(* IEC 61131-3 sources: AXOpen/src/abstractions/ctrl/src/Messaging/Dynamic, 9 files *)

(* ---- eAxoMessageDigestMethod.st ---- *)
NAMESPACE AXOpen.Messaging.Dynamic
    /// <summary>
    /// Message digest methods used to create fingerprint of a message.
    /// </summary>
    TYPE eAxoMessageDigestMethod : INT
    (
        /// <summary>
        /// Fastest method with highest probability of colisions.
        /// </summary>
        CRC8 := 8,

        /// <summary>
        /// Moderate speed method with lower probability of colisions.
        /// </summary>
        CRC16 := 16,

        /// <summary>
        /// Slowest speed method with relatively low probability of colisions.
        /// </summary>
        CRC32 := 32,

        /// <summary>
        /// Messages are not digested the repeated messages won't be filtered out.
        /// Use this option on low performance devices.
        /// </summary>
        NONE := 32767
    );
    END_TYPE
END_NAMESPACE

(* ---- IAxoMessageCategorize.st ---- *)
NAMESPACE AXOpen.Messaging.Dynamic
    INTERFACE IAxoMessageCategorize
		/// <summary>
        /// Categorizes and creates the message as 'debug'.
		/// </summary>
        METHOD AsDebug : IAxoMessageProperties END_METHOD

		/// <summary>
        /// Categorizes and creates the message as 'error'.
		/// </summary>
        METHOD AsError : IAxoMessageProperties END_METHOD

		/// <summary>
        /// Categorizes and creates the message as 'fatal'.
		/// </summary>
        METHOD AsFatal : IAxoMessageProperties END_METHOD

		/// <summary>
        /// Categorizes and creates the message as 'info'.
		/// </summary>
        METHOD AsInfo : IAxoMessageProperties END_METHOD

		/// <summary>
        /// Categorizes and creates the message as 'trace'.
		/// </summary>
        METHOD AsTrace : IAxoMessageProperties END_METHOD

		/// <summary>
        /// Categorizes and creates the message as 'warning'.
		/// </summary>
        METHOD AsWarning : IAxoMessageProperties END_METHOD
    END_INTERFACE
END_NAMESPACE

(* ---- IAxoMessageProperties.st ---- *)
NAMESPACE AXOpen.Messaging.Dynamic
    INTERFACE IAxoMessageProperties
        METHOD Pin: IAxoMessageProperties END_METHOD
        METHOD IsPinned: BOOL END_METHOD
    END_INTERFACE
END_NAMESPACE

(* ---- IAxoMessages.st ---- *)
NAMESPACE AXOpen.Messaging.Dynamic
    INTERFACE IAxoMessages
	    /// <summary>
		/// Adds message of 'debug' category to the message queue.
		/// </summary>
        METHOD Debug : IAxoMessageProperties
            VAR_INPUT
                /// <summary>
                /// Arbitrary message string.
                /// </summary>
                Message : STRING[AxoIntConstants#MAX_MESSAGE_TEXT_LENGHT];
            END_VAR
        END_METHOD

	    /// <summary>
		/// Adds message of 'error' category to the message queue.
		/// </summary>
        METHOD Error : IAxoMessageProperties
            VAR_INPUT
                /// <summary>
                /// Arbitrary message string.
                /// </summary>
                Message : STRING[AxoIntConstants#MAX_MESSAGE_TEXT_LENGHT];
            END_VAR
        END_METHOD

	    /// <summary>
		/// Adds message of 'information' category to the message queue.
		/// </summary>
        METHOD Info : IAxoMessageProperties
            VAR_INPUT
                /// <summary>
                /// Arbitrary message string.
                /// </summary>
                Message : STRING[AxoIntConstants#MAX_MESSAGE_TEXT_LENGHT];
            END_VAR
        END_METHOD

	    /// <summary>
		/// Adds message of 'notification' category to the message queue.
		/// </summary>
        METHOD Notify : IAxoMessageProperties
            VAR_INPUT
                /// <summary>
                /// Arbitrary message string.
                /// </summary>
                Message : STRING[AxoIntConstants#MAX_MESSAGE_TEXT_LENGHT];
            END_VAR
        END_METHOD

	    /// <summary>
		/// Adds message of 'programming error' category to the message queue.
		/// </summary>
        METHOD Programming : IAxoMessageProperties
            VAR_INPUT
                /// <summary>
                /// Arbitrary message string.
                /// </summary>
                Message : STRING[AxoIntConstants#MAX_MESSAGE_TEXT_LENGHT];
            END_VAR
        END_METHOD

	    /// <summary>
		/// Adds message of 'trace' category to the message queue.
		/// </summary>
        METHOD Trace : IAxoMessageProperties
            VAR_INPUT
                /// <summary>
                /// Arbitrary message string.
                /// </summary>
                Message : STRING[AxoIntConstants#MAX_MESSAGE_TEXT_LENGHT];
            END_VAR
        END_METHOD

	    /// <summary>
		/// Adds message of 'warning' category to the message queue.
		/// </summary>
        METHOD Warning : IAxoMessageProperties
            VAR_INPUT
                /// <summary>
                /// Arbitrary message string.
                /// </summary>
                Message : STRING[AxoIntConstants#MAX_MESSAGE_TEXT_LENGHT];
            END_VAR
        END_METHOD

        METHOD Build: IAxoMessageTextBuilder END_METHOD

        /// <summary>
		/// Adds message of given category to the message queue.
		/// </summary>
		/// <returns>Message index.</returns>
        METHOD Post  : IAxoMessageProperties
            VAR_INPUT
                /// <summary>
                /// Arbitrary message string.
                /// </summary>
                Message : STRING[AxoIntConstants#MAX_MESSAGE_TEXT_LENGHT];
                /// <summary>
                /// Message category.
                /// </summary>
                Category : eAxoMessageCategory;
            END_VAR
        END_METHOD

		/// <summary>
		/// Unpins this messenger.
		/// </summary>
        METHOD UnPin END_METHOD

    END_INTERFACE
END_NAMESPACE

(* ---- IAxoMessageTextBuilder.st ---- *)
NAMESPACE AXOpen.Messaging.Dynamic
    INTERFACE IAxoMessageTextBuilder
		/// <summary>
		/// Appends string to the message text.
		/// </summary>
		/// <remarks>
		/// 	<note type="warning">
		/// 		The size of the resulting string should not be more than '160' characters. The characters exceeding this size will be truncated.
		/// 	</note>
		/// </remarks>
 		METHOD Append : IAxoMessageTextBuilder VAR_INPUT Data : BOOL; END_VAR END_METHOD
		METHOD Append : IAxoMessageTextBuilder VAR_INPUT Data : BYTE; END_VAR END_METHOD
		METHOD Append : IAxoMessageTextBuilder VAR_INPUT Data : WORD; END_VAR END_METHOD
		METHOD Append : IAxoMessageTextBuilder VAR_INPUT Data : DWORD; END_VAR END_METHOD
		METHOD Append : IAxoMessageTextBuilder VAR_INPUT Data : LWORD; END_VAR END_METHOD
		METHOD Append : IAxoMessageTextBuilder VAR_INPUT Data : SINT; END_VAR END_METHOD
		METHOD Append : IAxoMessageTextBuilder VAR_INPUT Data : INT; END_VAR END_METHOD
		METHOD Append : IAxoMessageTextBuilder VAR_INPUT Data : DINT; END_VAR END_METHOD
		METHOD Append : IAxoMessageTextBuilder VAR_INPUT Data : LINT; END_VAR END_METHOD
		METHOD Append : IAxoMessageTextBuilder VAR_INPUT Data : USINT; END_VAR END_METHOD
		METHOD Append : IAxoMessageTextBuilder VAR_INPUT Data : UINT; END_VAR END_METHOD
		METHOD Append : IAxoMessageTextBuilder VAR_INPUT Data : UDINT; END_VAR END_METHOD
		METHOD Append : IAxoMessageTextBuilder VAR_INPUT Data : ULINT; END_VAR END_METHOD
		METHOD Append : IAxoMessageTextBuilder VAR_INPUT Data : REAL; END_VAR END_METHOD
		METHOD Append : IAxoMessageTextBuilder VAR_INPUT Data : LREAL; END_VAR END_METHOD
		METHOD Append : IAxoMessageTextBuilder VAR_INPUT Data : TIME; END_VAR END_METHOD
		METHOD Append : IAxoMessageTextBuilder VAR_INPUT Data : LTIME; END_VAR END_METHOD
		METHOD Append : IAxoMessageTextBuilder VAR_INPUT Data : DATE; END_VAR END_METHOD
		METHOD Append : IAxoMessageTextBuilder VAR_INPUT Data : LDATE; END_VAR END_METHOD
		METHOD Append : IAxoMessageTextBuilder VAR_INPUT Data : TIME_OF_DAY; END_VAR END_METHOD
		METHOD Append : IAxoMessageTextBuilder VAR_INPUT Data : LTIME_OF_DAY; END_VAR END_METHOD
		METHOD Append : IAxoMessageTextBuilder VAR_INPUT Data : DATE_AND_TIME; END_VAR END_METHOD
		METHOD Append : IAxoMessageTextBuilder VAR_INPUT Data : LDATE_AND_TIME; END_VAR END_METHOD
		METHOD Append : IAxoMessageTextBuilder VAR_INPUT Data : CHAR; END_VAR END_METHOD
		// METHOD Append : IAxoMessageTextBuilder VAR_INPUT Data : WCHAR; END_VAR END_METHOD
		METHOD Append : IAxoMessageTextBuilder VAR_INPUT Data : STRING[AxoIntConstants#MAX_MESSAGE_TEXT_LENGHT]; END_VAR END_METHOD
		// METHOD Append : IAxoMessageTextBuilder VAR_INPUT Data : WSTRING[IxIntConstants#MAX_MESSAGE_TEXT_LENGHT]; END_VAR END_METHOD
		/// <summary>
		/// Gets categorization methods for fluent message builder.
		/// </summary>
        METHOD As : IAxoMessageCategorize END_METHOD

		/// <summary>
		/// Initiates new message text building for this messenger in fluent-like fashion.
		/// </summary>
        METHOD Build : IAxoMessageTextBuilder END_METHOD
    END_INTERFACE
END_NAMESPACE

(* ---- IAxoMessenger.st ---- *)
NAMESPACE AXOpen.Messaging.Dynamic
    INTERFACE IAxoMessenger
		/// <summary>
		/// Clears the message content.
		/// <remarks>
		/// 	<note type="important">
		/// 		This method is exposed for Rpc calls, for testing purposes. Rpc calls of this method must not be used in production code
		///		</note>
		/// </remarks>
		/// </summary>
		METHOD Clear END_METHOD

		METHOD OnCondition : IAxoMessages
			VAR_INPUT
				inCondition : BOOL;
			END_VAR
		END_METHOD
    END_INTERFACE
END_NAMESPACE

(* ---- IAxoMessengerEnv.st ---- *)
NAMESPACE AXOpen.Messaging.Dynamic
    INTERFACE IAxoMessengerEnv
		/// <summary>
		/// Gets whether the messaging is suspended at this point in program.
		/// <para>
		/// See also <see cref="PlcDocu.TcoCore.TcoMessengerSettings.Resume()"/>
		/// </para>
		/// <para>
		/// See also <see cref="PlcDocu.TcoCore.TcoMessengerSettings.Suspend()"/>
		/// </para>
		/// <para>
		/// See also <see cref="PlcDocu.TcoCore.TcoMessengerSettings.MinLevel"/>
		/// </para>
		/// </summary>
		METHOD IsSuspended: BOOL END_METHOD
		/// <summary>
		/// Gets the message digest method.
		/// Message digest serves to fingerprint messages.
		/// </summary>
		METHOD GetMessageDigestMethod : eAxoMessageDigestMethod END_METHOD
		/// <summary>
		/// Sets the message digest method.
		/// Message digest serves to fingerprint messages.
		/// </summary>
		METHOD SetMessageDigestMethod VAR_INPUT inDigestMethod : eAxoMessageDigestMethod; END_VAR END_METHOD
		/// <summary>
		/// Gets the minimal messaging level, the objects will post only messages for the levels of this or superior severity.
		/// <para>
		/// See also <see cref="PlcDocu.TcoCore.TcoMessengerSettings.Resume()"/>
		/// </para>
		/// <para>
		/// See also <see cref="PlcDocu.TcoCore.TcoMessengerSettings.Suspend()"/>
		/// </para>
		/// <para>
		/// See also <see cref="PlcDocu.TcoCore.TcoMessengerSettings.MinLevel"/>
		/// </para>
		/// </summary>
		METHOD GetMinLevel : eAxoMessageCategory END_METHOD
		/// <summary>
		/// Sets the minimal messaging level, the objects will post only messages for the levels of this or superior severity.
		/// <para>
		/// See also <see cref="PlcDocu.TcoCore.TcoMessengerSettings.Resume()"/>
		/// </para>
		/// <para>
		/// See also <see cref="PlcDocu.TcoCore.TcoMessengerSettings.Suspend()"/>
		/// </para>
		/// <para>
		/// See also <see cref="PlcDocu.TcoCore.TcoMessengerSettings.MinLevel"/>
		/// </para>
		/// </summary>
		METHOD SetMinLevel VAR_INPUT inMessageCategory : eAxoMessageCategory; END_VAR END_METHOD
		/// <summary>
		/// Resumes messaging from the all objects of this context, when the messaging was previously suspended by ```Suspend``` method.
		/// <para>
		/// See also <see cref="PlcDocu.TcoCore.TcoMessengerSettings.Suspend()"/>
		/// </para>
		/// <para>
		/// See also <see cref="PlcDocu.TcoCore.TcoMessengerSettings.MinLevel"/>
		/// </para>
		/// </summary>
		METHOD Resume END_METHOD
		/// <summary>
		/// Suspends messaging from the all objects of this context that would occur from this point in the call tree.
		/// <para>
		/// See also <see cref="PlcDocu.TcoCore.TcoMessengerSettings.Resume()"/>
		/// </para>
		/// <para>
		/// See also <see cref="PlcDocu.TcoCore.TcoMessengerSettings.MinLevel"/>
		/// </para>
		/// </summary>
		METHOD Suspend END_METHOD
	END_INTERFACE
END_NAMESPACE

(* ---- AxoMessageDigest.st ---- *)
NAMESPACE AXOpen.Messaging.Dynamic
    CLASS PUBLIC AxoMessageDigest
        VAR PUBLIC
            Digest : DWORD;
            Cycle : ULINT;
            Count : ULINT;
            Category : eAxoMessageCategory;
        END_VAR
    END_CLASS
END_NAMESPACE

(* ---- AxoMessengerEnv.st ---- *)
USING AXOpen.Utils;

NAMESPACE AXOpen.Messaging.Dynamic
    CLASS PUBLIC AxoMessengerEnv IMPLEMENTS IAxoMessengerEnv
		VAR
			_minLevel : eAxoMessageCategory;
			_isMessagingSuspended : BOOL;
			_messageDigestMethod : eAxoMessageDigestMethod := eAxoMessageDigestMethod#CRC16;
			//_messengerLoggingMethod : eIxMessengerLogMethod := eIxMessengerLogMethod#OnEventRisen;
			_sb : REF_TO AxoStringBuilder;
		END_VAR

		/// <inheritdoc />
		METHOD PUBLIC IsSuspended: BOOL
			IsSuspended := _isMessagingSuspended;
		END_METHOD

		/// <inheritdoc />
		METHOD PUBLIC GetMessageDigestMethod : eAxoMessageDigestMethod
			GetMessageDigestMethod := _messageDigestMethod;
		END_METHOD

		/// <inheritdoc />
		METHOD PUBLIC SetMessageDigestMethod
			VAR_INPUT
				inDigestMethod : eAxoMessageDigestMethod;
			END_VAR
			_messageDigestMethod := inDigestMethod;
		END_METHOD

		/// <inheritdoc />
		METHOD PUBLIC GetMinLevel : eAxoMessageCategory
			GetMinLevel := _minLevel;
		END_METHOD

		/// <inheritdoc />
		METHOD PUBLIC SetMinLevel
			VAR_INPUT
				inMessageCategory : eAxoMessageCategory;
			END_VAR
			_minLevel := inMessageCategory;
		END_METHOD

		/// <inheritdoc />
		METHOD PUBLIC Resume
			_isMessagingSuspended := FALSE;
		END_METHOD

		/// <inheritdoc />
		METHOD PUBLIC Suspend
			_isMessagingSuspended := TRUE;
		END_METHOD

		/// <inheritdoc />
		METHOD PUBLIC GetStringBuilder : REF_TO AxoStringBuilder
			GetStringBuilder ?= _sb;
		END_METHOD
	END_CLASS
END_NAMESPACE
